FUNCTION_BLOCK PROGERRCTRL_DEB (* Corrects forecast errors of the BatteryOptimizer FB. *)
  (* Standard: 61499-2; Description: IEC 61499 implementation of the "PVprog" algorithm. Original version's MIT license: Copyright (c) 2016 Joseph Bergner, Johannes Weniger, Tjarko Tjaden Permission is hereby granted, free of charge, to any person obtaining a copy of this software and associated documentation files (the "Software"), to deal in the Software without restriction, including without limitation the rights to use, copy, modify, merge, publish, distribute, sublicense, and/or sell copies of the Software, and to permit persons to whom the Software is furnished to do so, subject to the following conditions: The above copyright notice and this permission notice shall be included in all copies or substantial portions of the Software. THE SOFTWARE IS PROVIDED "AS IS", WITHOUT WARRANTY OF ANY KIND, EXPRESS OR IMPLIED, INCLUDING BUT NOT LIMITED TO THE WARRANTIES OF MERCHANTABILITY, FITNESS FOR A PARTICULAR PURPOSE AND NONINFRINGEMENT. IN NO EVENT SHALL THE AUTHORS OR COPYRIGHT HOLDERS BE LIABLE FOR ANY CLAIM, DAMAGES OR OTHER LIABILITY, WHETHER IN AN ACTION OF CONTRACT, TORT OR OTHERWISE, ARISING FROM, OUT OF OR IN CONNECTION WITH THE SOFTWARE OR THE USE OR OTHER DEALINGS IN THE SOFTWARE. *)
  (* Version 1.0, 2017-05-22, Marc Jakobi, HTW Berlin *)
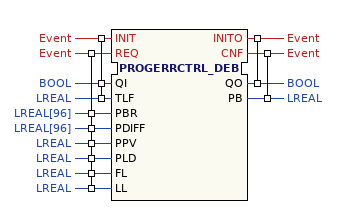
  EVENT_INPUT
    INIT WITH QI, TLF; (* Initialization Request *)
    REQ WITH PBR, PPV, PLD, LL, FL, PDIFF; (* Normal Execution Request *)
  END_EVENT
  EVENT_OUTPUT
    INITO WITH QO; (* Initialization Confirm *)
    CNF WITH PB; (* Execution Confirmation *)
  END_EVENT
  VAR_INPUT
    QI : BOOL; (* Input event qualifier *)
    TLF : LREAL := 15; (* Time frame forecasted ahead (looked forward) in h *)
    PBR : ARRAY [0..95] OF LREAL; (* Battery charge (positive)/discharge (negative) roadmap (power in W) over the forecast horizon *)
    PDIFF : ARRAY [0..95] OF LREAL; (* Power difference forecast in W (negative = PV deficit, positive = PV surplus) *)
    PPV : LREAL; (* Current PV power in W *)
    PLD : LREAL; (* Current load in W *)
    FL : LREAL; (* Feed-in limitation in W (0 for none) *)
    LL : LREAL; (* Load limit in W (0 for none) *)
  END_VAR
  VAR_OUTPUT
    QO : BOOL; (* Output event qualifier *)
    PB : LREAL; (* Set battery charging power in W (positive = charge, negative = discharge) *)
  END_VAR
  VAR
    LOOKFORWARDTIMEINTIMESTEPS : UINT := 60; (* Number of time steps (15 min intervals) to look ahead for forecast *)
    PDIFFC : LREAL; (* Current power difference (PPV - PLD) *)
    CCFLAG : BOOL; (* Flag to check control conditions *)
    LIMITCHK : LREAL; (* Limit (feed-in or load) to check control condition against *)
    BCDFLAG : BOOL; (* Flag to check whether battery charging (true) or discharging (false) needs to be corrected *)
  END_VAR
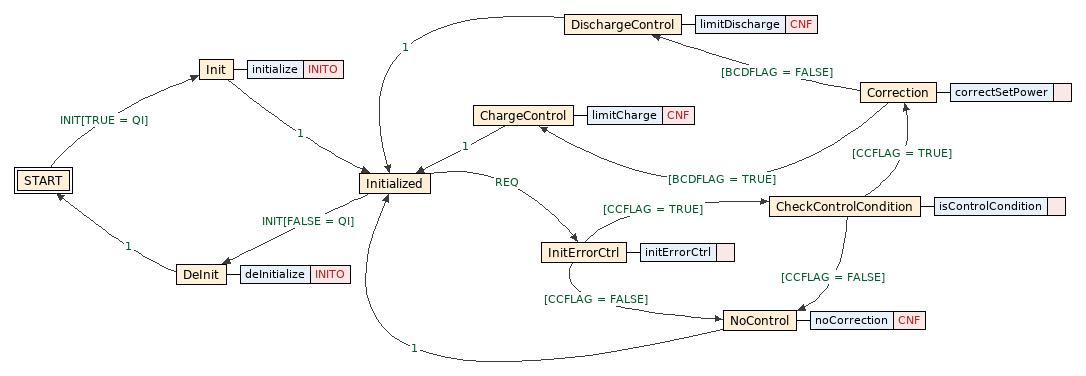
  EC_STATES
    START; (* Initial State *)
    Init : initialize -> INITO; (* Initialization *)
    InitErrorCtrl : initErrorCtrl; (* Normal execution *)
    Initialized;
    DeInit : deInitialize -> INITO;
    CheckControlCondition : isControlCondition;
    NoControl : noCorrection -> CNF;
    ChargeControl : limitCharge -> CNF;
    DischargeControl : limitDischarge -> CNF;
    Correction : correctSetPower;
  END_STATES
  EC_TRANSITIONS
    START TO Init := INIT[TRUE = QI];
    Init TO Initialized := 1;
    Initialized TO InitErrorCtrl := REQ;
    DeInit TO START := 1;
    Initialized TO DeInit := INIT[FALSE = QI];
    InitErrorCtrl TO CheckControlCondition := [CCFLAG = TRUE];
    CheckControlCondition TO NoControl := [CCFLAG = FALSE];
    NoControl TO Initialized := 1;
    ChargeControl TO Initialized := 1;
    DischargeControl TO Initialized := 1;
    CheckControlCondition TO Correction := [CCFLAG = TRUE];
    Correction TO DischargeControl := [BCDFLAG = FALSE];
    Correction TO ChargeControl := [BCDFLAG = TRUE];
    InitErrorCtrl TO NoControl := [CCFLAG = FALSE];
  END_TRANSITIONS
  ALGORITHM initialize IN ST: (* Initialization algorithm *)
VAR
	tmp1 : LREAL;
	tmp2 : UINT;
END_VAR;
/*
 * Used internal vars & inputs:
 * TLF, LOOKFORWARDTIMEINTIMESTEPS : UINT;
 */
tmp1 := TLF * 4; // output resolution = 15 min
tmp2 := LREAL_TO_UINT(tmp1);
IF UINT_TO_LREAL(tmp2) < tmp1 THEN
 	LOOKFORWARDTIMEINTIMESTEPS := tmp2 + 1;
ELSE
	LOOKFORWARDTIMEINTIMESTEPS := tmp2;
END_IF;
// Set output event qualifier
QO := QI;
  END_ALGORITHM
  ALGORITHM deInitialize IN ST: (* Normally executed algorithm *)
QO := FALSE;
  END_ALGORITHM
  ALGORITHM initErrorCtrl IN ST: (* Initializes variables for error control *)
/*
 * Used internal vars & inputs:
 * PDIFFC, PPV, PLD, FL, LL, LIMITCHK : LREAL;
 * CCFLAG, BCDFLAG : BOOL;
 */
PDIFFC := PPV - PLD;
IF (PDIFFC > 0 AND FL <> 0) THEN // Surplus power  & PV feed-in limitation
	LIMITCHK := FL;
	CCFLAG := TRUE;
	BCDFLAG := TRUE;
ELSIF (PDIFFC < 0 AND LL <> 0) THEN // Power deficit and load peak shaving
	LIMITCHK := LL;
	CCFLAG := TRUE;
	BCDFLAG := FALSE;
ELSE // No control necessary
	CCFLAG := FALSE;
END_IF;
  END_ALGORITHM
  ALGORITHM isControlCondition IN ST: (* Checks whether control is necessary or not *)
VAR
	cond1 : BOOL;
	cond2 : BOOL;
	cond3 : BOOL;
	maxDif : LREAL;
	absPDF : LREAL;
	absBCR : LREAL;
	absPDFC : LREAL;
	i : UINT;
END_VAR;
/*
 * Used internal vars & inputs:
 * PBR,PDIFF, PDIFFC, LIMITCHK : LREAL;
 * CCFLAG : BOOL;
 */
cond1 := FALSE;
cond2 := FALSE;
cond3 := FALSE;
// Condition 1: The forecasted charging or discharging power for the current time step is not zero
IF PBR[0] <> 0 THEN
	cond1 := TRUE;
END_IF;
/*
 * Condition 2: The current forecasted power difference [PPV-PLD] is greater than the maximum of the predicted
 * feed-in power over the forecast horizon.
 */
maxDif := 0;
FOR i := 0 TO LOOKFORWARDTIMEINTIMESTEPS - 1 BY 1 DO
	absPDF := PDIFF[i]; // ABS(PDIFF)
	IF absPDF < 0 THEN
		absPDF := absPDF * (-1);
	END_IF;
	absBCR := PBR[i];  // ABS(PBR)
	IF absBCR < 0 THEN
		absBCR := absBCR * (-1);
	END_IF;
	IF absPDF - absBCR > maxDif THEN
		maxDif := absPDF - absBCR;
	END_IF;
END_FOR;
IF PDIFFC >= 0 THEN // ABS(PDIFFC)
	absPDFC := PDIFFC;
ELSE
	absPDFC := PDIFFC * (-1);
END_IF;
IF absPDFC > maxDif THEN
	cond2 := TRUE;
END_IF;
// Condition 3: The current power difference is greater than the maximum permissible feed-in limitation
IF LIMITCHK < 0 THEN
	LIMITCHK := LIMITCHK * (-1);
END_IF;
IF absPDFC > LIMITCHK THEN
	cond3 := TRUE;
END_IF;
IF (cond1 OR cond2 OR cond3) THEN
	CCFLAG := TRUE;
ELSE
	CCFLAG := FALSE;
	PDIFFC := 0; // Set charging/discharging power to zero to prevent stepped adjustment
END_IF;
  END_ALGORITHM
  ALGORITHM noCorrection IN ST: (* Sets the battery charge without correcting errors *)
PB := PDIFFC;
  END_ALGORITHM
  ALGORITHM limitCharge IN ST: (* Limits charging power to zero and greater *)
IF PB < 0 THEN
	PB := 0;
END_IF;
  END_ALGORITHM
  ALGORITHM limitDischarge IN ST: (* Limits discharging power to zero and below *)
IF PB > 0 THEN
	PB := 0;
END_IF;
  END_ALGORITHM
  ALGORITHM correctSetPower IN ST: (* Corrects the set power according to forecast error *)
PB := PBR[0] + PDIFFC - PDIFF[0];
  END_ALGORITHM
END_FUNCTION_BLOCK
